// TIA Portal V18 export
VAR_GLOBAL   // PLC tag table "Default tag table"
   btn_1 AT %I0.0 : Bool;
END_VAR
